// TwinCAT 3 PLC project PLC_Refrigirator_prj_ST
// ProgramVersion: 3.1.4023.0
// libraries:
//   Tc2_Standard, * (Beckhoff Automation GmbH)
//   Tc2_System, * (Beckhoff Automation GmbH)
//   Tc3_Module, * (Beckhoff Automation GmbH)
//   VisuDialogs, * (System)
//   VisuSymbols,3.5.10.0,System
// project tree:
//   / GlobalTextList.TcGTLO, PlcTask.TcTTO, Visualisierungsmanager.TcVMO (not stored)
//   GVLs/ GVL_Var.TcGVL
//   POUs/ FB_Blinker1.TcPOU, MAIN.TcPOU, Signal1.TcPOU, Simulation.TcPOU
//   VISUs/ Visualization.TcVIS
// real-time tasks:
//   TASK PlcTask: cycle T#10ms, priority 20, ADS port 350

CONFIGURATION PLC_Refrigirator_prj_ST
    RESOURCE PLC ON TwinCAT3
        TASK PlcTask(INTERVAL := T#10ms, PRIORITY := 20);
        PROGRAM Simulation WITH PlcTask : Simulation;
        PROGRAM MAIN WITH PlcTask : MAIN;
    END_RESOURCE
END_CONFIGURATION

// ---- GVLs/GVL_Var.TcGVL
{attribute 'qualified_only'}
VAR_GLOBAL
	bDoorOpen: BOOL := FALSE;
	fTempSet: REAL := 8.0;
	fTempActual: REAL := 8.0;
	bCompressor: BOOL := FALSE;
	tDoorOpenThreshold: TIME := T#10s;
	tlmAlaramThreshold: TIME := T#30s;
	bSignal: BOOL := FALSE;
	bLamp: BOOL := FALSE;
END_VAR

// ---- POUs/Simulation.TcPOU
PROGRAM Simulation
VAR
	fbT1				: TON;				//The temperature is decreased on a time dalay
	tCooling			: TIME := T#500MS;	//Cooling rate
	bReduceTemp			: BOOL;				//Signal for decreasing the temperature
	fbT2				: TON;				//The temperature is increased on a time delay
	tEnvironment		: TIME := T#2S;		//Delay time when the door is closed
	tEnvironmentDoorOpen: TIME := T#1S;		//Delay time when the door is open
	bRaiseTemp			: BOOL;				//Signal for increasing the temperature
	tImTemp				: TIME;				//Delay time
	nCounter			: INT;				//Iteration of the programm
END_VAR

//After the compressor has been activated due to fTempActual being too high, the temperature decreases.
//The temperature is decreased by 0.1°C per cycle after a delay of P_Cooling
IF GVL_VAR.bCompressor THEN
	fbT1(IN:= GVL_VAR.bCompressor, PT:= tCooling, Q=> bReduceTemp);
	IF bReduceTemp THEN
		GVL_VAR.fTempActual:= GVL_VAR.fTempActual-0.1;
		fbT1(IN:= FALSE);
	END_IF
END_IF

//If the door is open, the warming will occur faster; SEL chooses between tEnvironment or tEnvironmentDoorOpen
tImTemp:= SEL(GVL_VAR.bDoorOpen, tEnvironment, tEnvironmentDoorOpen);

//If the compressor is not in operation, then the cooling chamber will become warmer.
//The temperature is incremental by 0.1°C per cycle after a delay of tImTemp
fbT2(IN:= TRUE, PT:= tImTemp, Q=> bRaiseTemp);
IF bRaiseTemp THEN
	GVL_VAR.fTempActual:= GVL_VAR.fTempActual+0.1;
	fbT2(IN:= FALSE);
END_IF

nCounter := nCounter+1;

END_PROGRAM

// ---- POUs/MAIN.TcPOU
PROGRAM MAIN
VAR
	fHysteresis: REAL := 1;		//Hysteresis value
	rUpperLimit: REAL;		 	//Temperature set value added with Hysteresis
	rLowerLimit: REAL;		 	//Temperature set value subtracted with Hysteresis
END_VAR

rUpperLimit := GVL_Var.fTempSet + fHysteresis;
rLowerLimit := GVL_Var.fTempSet - fHysteresis;

// Logic to switch ON the compressor when it exceeds the UpperLimit
// and compressor switched OFF when it is below the lowerLimit
IF GVL_Var.fTempActual > rUpperLimit THEN
	GVL_Var.bCompressor := TRUE;
ELSIF GVL_Var.fTempActual < rLowerLimit THEN
	GVL_Var.bCompressor := FALSE; 
END_IF

//Calling Signal1 Program
Signal1();

END_PROGRAM

// ---- POUs/Signal1.TcPOU
PROGRAM Signal1
VAR
	fbTimer1: TON;			//Timer1 Initialization
	fbTimer2: TON;			//Timer2 Initialization
	Blinker: FB_Blinker1;	//Function Block Blinker1 Initialization
END_VAR

//Timer1 Parameterization
fbTimer1(IN := GVL_Var.bCompressor,
		PT	:= GVL_Var.tlmAlaramThreshold,
		Q	=> GVL_Var.bSignal
		);
//Timer2 Parameterization
fbTimer2(IN := GVL_Var.bDoorOpen,
		PT	:= GVL_Var.tlmAlaramThreshold
		);
//Blinker Parameterization	
Blinker(bStart := fbTimer2.Q,
		tSignalTimeOff := T#1S, 
		tSignalTimeOn	:= T#1S,
		bOut => GVL_Var.bSignal );
//To switch ON the Lamp when Door is open		
IF GVL_Var.bDoorOpen THEN
	GVL_Var.bLamp := TRUE;
ELSIF NOT GVL_Var.bDoorOpen THEN
	GVL_Var.bLamp := FALSE;
END_IF

END_PROGRAM

// ---- POUs/FB_Blinker1.TcPOU
FUNCTION_BLOCK FB_Blinker1
VAR_INPUT
	bStart: BOOL;         	//Start signal 
	tSignalTimeOn: TIME;  	//Pulse Time On
	tSignalTimeOff: TIME;	//Pulse Time Off
END_VAR
VAR_OUTPUT
	bOut: BOOL;				//Output pulse 
END_VAR
VAR
	fbTimerA: TON;			//TimerA Initialization
	fbTimerB: TON;			//TimerB Initialization
END_VAR

// Timer A Parameterization
fbTimerA(IN := (bStart AND NOT fbTimerB.Q),
		PT := tSignalTimeOn,
		Q => bOut
		);

// Timer B Parameterization	
fbTimerB(IN := fbTimerA.Q,
		PT := tSignalTimeOff,
		);

END_FUNCTION_BLOCK

// ---- GlobalTextList.TcGTLO
TEXTLIST GlobalTextList
  629 = 'Actual Temperature'
  462 = 'Enter the Set Value'
  30 = 'Fridge Lamp which light the Interior'
  366 = 'Handle to open Fridge Door'
  845 = 'Indicates when Fridge Door opened for long time'
  895 = 'njjjjj'
  253 = 'Set Temp'
  274 = 'Set the Actual Temp'
  745 = 'Set the Temp to be maintained in Fridge between 0 and 20'
  641 = 'State of Compressor'
END_TEXTLIST

// ---- VISUs/Visualization.TcVIS
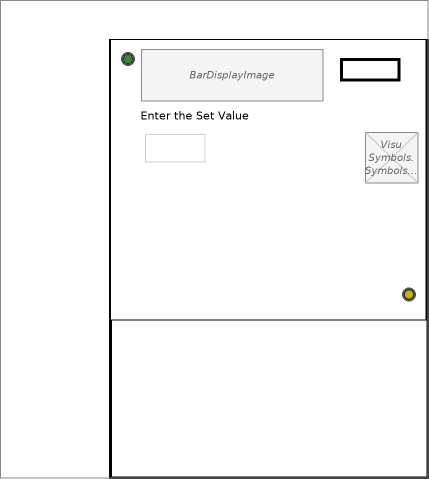
VISUALIZATION Visualization  // 429x479
    Rectangle (109,39 320x440)
    Rectangle (110,39 316x281)
    RoundedRectangle (340,58 60x23), tooltip "Handle to open Fridge Door"
        OnMouseClick: toggle GVL_Var.bDoorOpen
    Image (365,132 53x51), angle 182, tooltip "Fridge Lamp which light the Interior", invisible if: NOT GVL_Var.bLamp, image: VisuSymbols.Symbols.light
        p2175578022: GVL_Var.bLamp
    Textfield (145,134 60x28), tooltip "Set the Temp to be maintained in Fridge between 0 and 20", text variable: GVL_Var.fTempSet
        OnMouseClick: write the text variable via Default, min 0, max 20
    Lamp1 (401,283 16x23), tooltip "Indicates when Fridge Door opened for long time", variable: GVL_Var.bSignal, style: Lamp-Lamp1-Yellow
    Lamp1 (120,49 16x20), tooltip "State of Compressor", variable: GVL_Var.bCompressor, style: Lamp-Lamp1-Green
    BarDisplayImage (141,49 182x52), value: GVL_Var.fTempActual, style: BarDisplayImage-Gray, scale format: %.1f, scale 0..20
    Label (120,101 150x30), "Enter the Set Value"
END_VISUALIZATION
